FUNCTION_BLOCK INTEGRATOR
  (* Standard: 61499-2 *)
  (* Version 15-04-2013, Gabriel *)
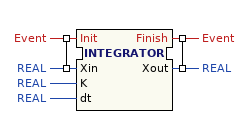
  EVENT_INPUT
    Init WITH Xin;
  END_EVENT
  EVENT_OUTPUT
    Finish WITH Xout;
  END_EVENT
  VAR_INPUT
    Xin : REAL;
    K : REAL;
    dt : REAL;
  END_VAR
  VAR_OUTPUT
    Xout : REAL;
  END_VAR
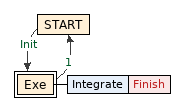
  EC_STATES
    Exe : Integrate -> Finish;
    START;
  END_STATES
  EC_TRANSITIONS
    Exe TO START := 1;
    START TO Exe := Init;
  END_TRANSITIONS
  ALGORITHM Integrate IN Lua:
Xout = Xout + K*dt*Xin
  END_ALGORITHM
END_FUNCTION_BLOCK
